TYPE DUT_HMI_00_MANUALS :
STRUCT
	PS : ARRAY[0..CNC.NUM_MAX_MANUALS_00-1] OF BOOL;
	LS : ARRAY[0..CNC.NUM_MAX_MANUALS_00-1] OF BOOL;
END_STRUCT
END_TYPE

(* stored: Version 1.1.0.1, ProductVersion 3.1.4024.13
   DUT DUT_HMI_00_MANUALS: Id {0ac636ad-71b2-4bba-900e-3a66facc286a} *)
